SUBAPPLICATION logiBUS_AI_Calibrate_Remote_IDA_OPC (* 2-Punkt-Kalibrierung (AR_CALIBRATE_2P_REF, unabhaengig gespeicherte Rohwerte X_LOW/X_HIGH + Referenzwerte LOW_REF/HIGH_REF alle INI-persistiert) auf VT-Zahlenfelder (Rohwert + kalibrierter Wert, je eigene CNumberVariable) + Bargraph (kalibriert) + 2 VT-Tasten (CO/CS) + OPC-UA (Rohwert DWORD + kalibrierter Wert REAL, generisch, ein Kanal). Wie logiBUS_AI_Calibrate_IDA_OPC, aber der Rohwert kommt per Remote-Subscribe (AD_SUBSCRIBE_1) statt von einem lokalen logiBUS_AI_IDA - fuer Sensoren, deren physischer Analog-Eingang auf einer Station OHNE VT-Anschluss sitzt (z.B. Schnitthoehen-Winkelsensor B13 auf APIXON STG3, waehrend Kalibrierung+VT auf der Station mit VT-Anschluss laufen). Der Rohwert wird dort per logiBUS_AI_Raw_Publish_OPC publiziert. *)
  (* Standard: 61499-2; Description: Copyright (c) 2026 Meisterschulen am Ostbahnhof This program and the accompanying materials are made available under the terms of the Eclipse Public License 2.0 which is available at https://www.eclipse.org/legal/epl-2.0/ SPDX-License-Identifier: EPL-2.0 *)
  (* Version 1.0, 2026-09-12, Franz Höpfinger, Meisterschulen am Ostbahnhof, Remote-Rohwert-Variante von logiBUS_AI_Calibrate_IDA_OPC - logiBUS_AI_IDA+AD_SPLIT_2+AD_PUBLISH_RAW durch AD_SUBSCRIBE_1 ersetzt, Rest der Kalibrier-/VT-Kette unveraendert. Fuer Schnitthoehen-Winkelsensor B13 (STG3), Kalibrierung+VT auf STG1. *)
  (* Version 1.1, 2026-09-17, Franz Höpfinger, Meisterschulen am Ostbahnhof, AR_CALIBRATE_2P_REF.C_LOW/C_HIGH von AX-Sockets auf reine EventInputs umgestellt (Franz-Entscheidung, siehe logiBUS_AI_Calibrate_IDA_OPC v1.3) - AX_BOOL_TO_X_CO/_CS entfallen ersatzlos, E_MERGE_CO_B/E_MERGE_CS_B verbinden jetzt direkt per EventConnection mit CALIBRATE.C_LOW/C_HIGH. Dieser Typ ist ohnehin durch logiBUS_AI_Calibrated_Subscribe_VT_OPC (Analog-Lokal-Verarbeitung, Plan cuddly-bubbling-twilight) auf dem Weg zur Ablösung - Anpassung hier nur, damit die Datei weiterhin kompiliert. *)
  (* Version 1.2, 2026-09-18, Franz Höpfinger, Meisterschulen am Ostbahnhof, CO/CS-Merge-Ketten (2x E_MERGE_2 in Reihe) durch je einen einzelnen E_MERGE_3 ersetzt - OR-Merge ist assoziativ, funktional identisch. Siehe logiBUS_AI_Calibrate_IDA_OPC v1.4. *)
  (* Version 1.4, 2026-09-21, Franz Höpfinger, Meisterschulen am Ostbahnhof, Code-Review-Fund (PR #260): INI_X_HIGH.DEFAULT_VALUE stand auf REAL#1.0 statt 0.0 - AR_CALIBRATE_2P_REF's xHighCal-Kalibriert-Flag latchte dadurch bei JEDEM Boot sofort TRUE, obwohl HIGH nie kalibriert wurde. Default auf REAL#0.0 korrigiert. Betrifft Schnitthoehe/Oeltemperatur/Druck. *)
  (* Version 1.3, 2026-09-21, Franz Höpfinger, Meisterschulen am Ostbahnhof, AR_CALIBRATE_2P_REF hat jetzt ein INIT/QI/QO-Enable-Pattern (Bugfix Garbage-Interpolation bei nur einem kalibrierten Punkt + xClipping) - CALIBRATE bekommt Parameter QI=TRUE, sonst bleibt die FB im START-Zustand haengen und REQ laeuft nie. *)
  PACKAGE MyLib::sys;
  IMPORT isobus::UT::Q::const::IDs::ID_NULL;
  IMPORT logiBUS::utils::conversion::phys::NumericObjectPool_S;
  IMPORT isobus::UT::io::Button::ButtonActivationCode::BT_PRESSED_LATCHED;
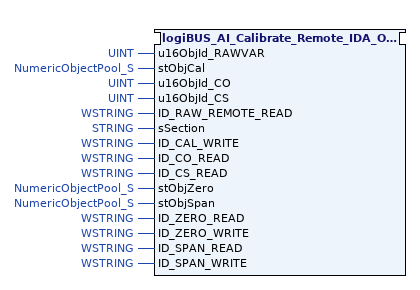
  VAR_INPUT
    u16ObjId_RAWVAR : UINT := ID_NULL; (* Object ID CNumberVariable (Rohwert 0-4095, unkalibriert, reine Diagnose-Anzeige) *)
    stObjCal : logiBUS::utils::conversion::phys::NumericObjectPool_S := (u16ObjId := ID_NULL, r32Scale := 1.0, i32Offset := 0, u8Decimals := 1); (* Object ID + Scale/Offset/Decimals CNumberVariable (kalibrierter Wert, eigene, unabhaengige CNumberVariable) *)
    u16ObjId_CO : UINT := ID_NULL; (* Object ID Taste 'CO' (Kalibrier-Nullpunkt: Referenz 1 anlegen, dann druecken) *)
    u16ObjId_CS : UINT := ID_NULL; (* Object ID Taste 'CS' (Kalibrier-Spanne: Referenz 2 anlegen, dann druecken - erst nach CO moeglich) *)
    ID_RAW_REMOTE_READ : WSTRING; (* Remote-Subscribe-Adresse des Rohwerts (DWORD 0-4095, ACTION=SUBSCRIBE) - Gegenstueck zu ID_RAW_WRITE auf der Sensor-Station (logiBUS_AI_Raw_Publish_OPC) *)
    sSection : STRING; (* INI-Sektionsname fuer X_LOW/X_HIGH/LOW_REF/HIGH_REF-Persistenz - pro Kanal eindeutig, sonst kollidieren die Kanaele in settings.ini *)
    ID_CAL_WRITE : WSTRING; (* Kalibrierter-Wert-Ruckmelde-Adresse (REAL, ACTION=PUBLISH) *)
    ID_CO_READ : WSTRING; (* Remote-CO-Adresse (BOOL, ACTION=SUBSCRIBE, togglet Kalibrier-Nullpunkt-Trigger wie ein Tastendruck - Web-Client schreibt bei jedem Klick den invertierten letzten Wert, jede Flanke (steigend ODER fallend) loest CO aus) *)
    ID_CS_READ : WSTRING; (* Remote-CS-Adresse (BOOL, ACTION=SUBSCRIBE, togglet Kalibrier-Spanne-Trigger wie ein Tastendruck - siehe ID_CO_READ) *)
    stObjZero : logiBUS::utils::conversion::phys::NumericObjectPool_S := (u16ObjId := ID_NULL, r32Scale := 1.0, i32Offset := 0, u8Decimals := 1); (* Object ID + Scale/Offset/Decimals CNumberVariable (ZERO-Referenzwert, VT-Eingabefeld + OPC-UA) *)
    stObjSpan : logiBUS::utils::conversion::phys::NumericObjectPool_S := (u16ObjId := ID_NULL, r32Scale := 1.0, i32Offset := 0, u8Decimals := 1); (* Object ID + Scale/Offset/Decimals CNumberVariable (SPAN-Referenzwert, VT-Eingabefeld + OPC-UA) *)
    ID_ZERO_READ : WSTRING; (* Remote-Subscribe-Adresse ZERO-Referenzwert (REAL, ACTION=SUBSCRIBE) *)
    ID_ZERO_WRITE : WSTRING; (* Remote-Echo-Adresse ZERO-Referenzwert (REAL, ACTION=PUBLISH) *)
    ID_SPAN_READ : WSTRING; (* Remote-Subscribe-Adresse SPAN-Referenzwert (REAL, ACTION=SUBSCRIBE) *)
    ID_SPAN_WRITE : WSTRING; (* Remote-Echo-Adresse SPAN-Referenzwert (REAL, ACTION=PUBLISH) *)
  END_VAR
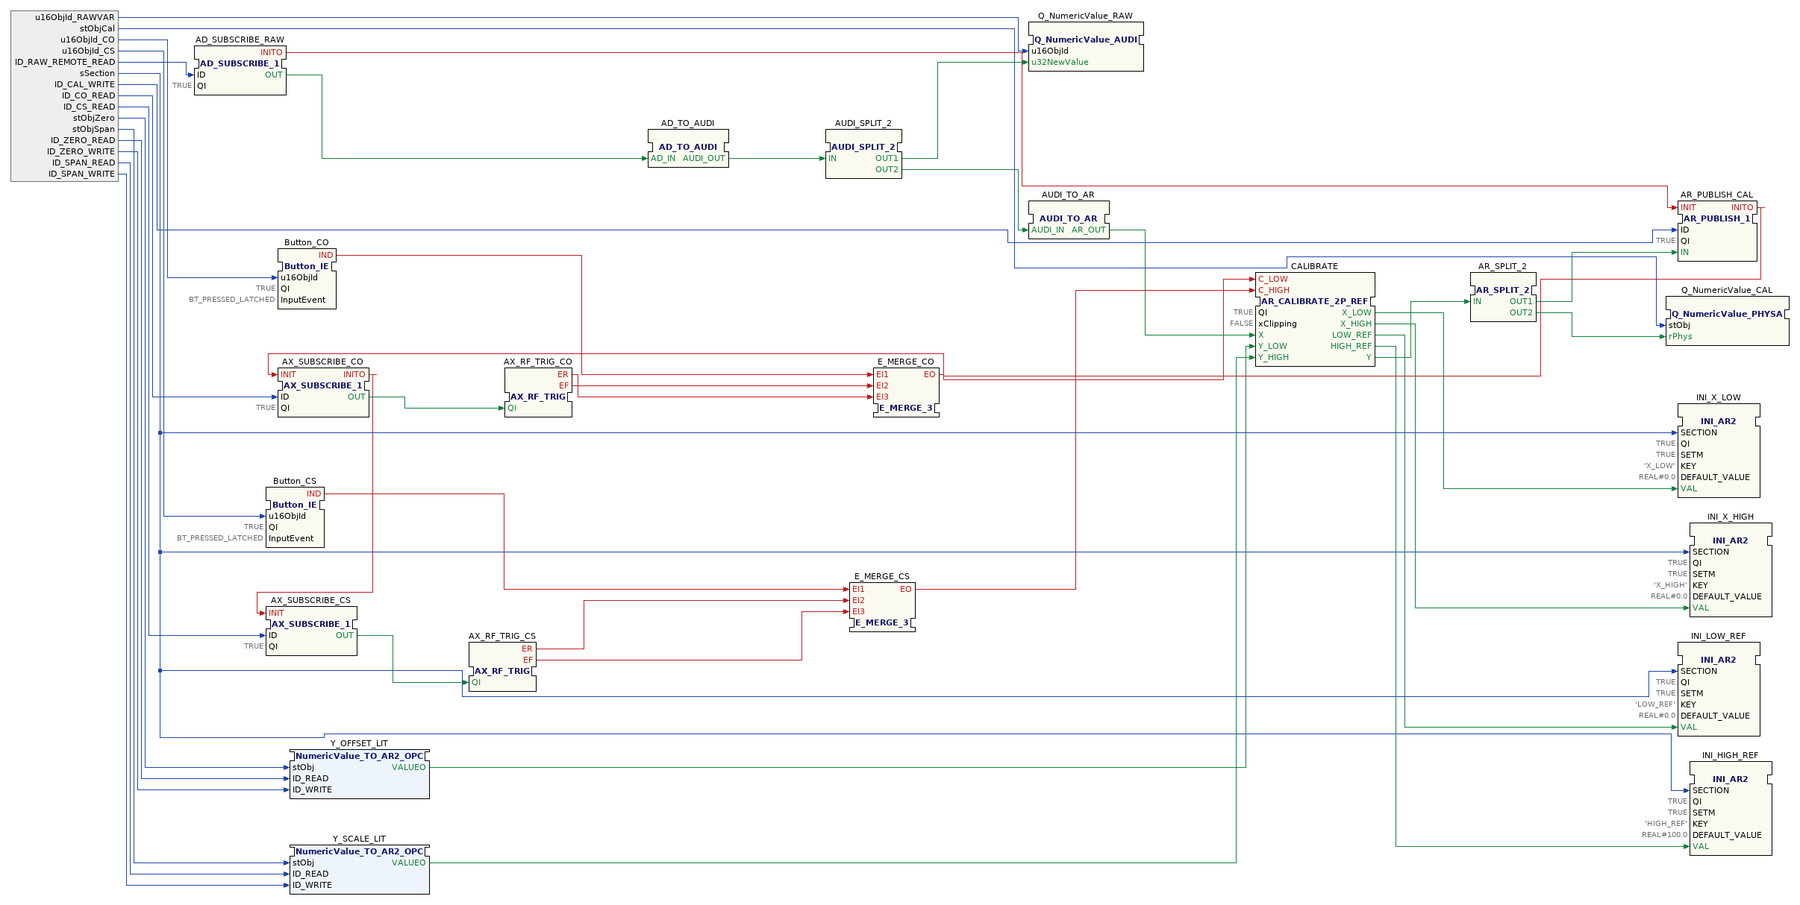
  FBS
    AD_SUBSCRIBE_RAW : adapter::net::AD_SUBSCRIBE_1(QI := TRUE);
    AD_TO_AUDI : adapter::conversion::unidirectional::AD_TO_AUDI;
    AUDI_SPLIT_2 : adapter::events::unidirectional::AUDI_SPLIT_2;
    Q_NumericValue_RAW : isobus::UT::Q::Q_NumericValue_AUDI;
    AUDI_TO_AR : adapter::conversion::unidirectional::AUDI_TO_AR;
    CALIBRATE : adapter::Engineering::measurements::AR_CALIBRATE_2P_REF(QI := TRUE, xClipping := FALSE);
    Button_CO : isobus::UT::io::Button::Button_IE(QI := TRUE, InputEvent := BT_PRESSED_LATCHED);
    Button_CS : isobus::UT::io::Button::Button_IE(QI := TRUE, InputEvent := BT_PRESSED_LATCHED);
    AX_SUBSCRIBE_CO : adapter::net::AX_SUBSCRIBE_1(QI := TRUE);
    AX_RF_TRIG_CO : adapter::events::unidirectional::AX_RF_TRIG;
    E_MERGE_CO : iec61499::events::E_MERGE_3;
    AX_SUBSCRIBE_CS : adapter::net::AX_SUBSCRIBE_1(QI := TRUE);
    AX_RF_TRIG_CS : adapter::events::unidirectional::AX_RF_TRIG;
    E_MERGE_CS : iec61499::events::E_MERGE_3;
    INI_X_LOW : eclipse4diac::storage::INI_AR2(QI := TRUE, SETM := TRUE, KEY := 'X_LOW', DEFAULT_VALUE := REAL#0.0);
    INI_X_HIGH : eclipse4diac::storage::INI_AR2(QI := TRUE, SETM := TRUE, KEY := 'X_HIGH', DEFAULT_VALUE := REAL#0.0);
    INI_LOW_REF : eclipse4diac::storage::INI_AR2(QI := TRUE, SETM := TRUE, KEY := 'LOW_REF', DEFAULT_VALUE := REAL#0.0);
    INI_HIGH_REF : eclipse4diac::storage::INI_AR2(QI := TRUE, SETM := TRUE, KEY := 'HIGH_REF', DEFAULT_VALUE := REAL#100.0);
    AR_SPLIT_2 : adapter::events::unidirectional::AR_SPLIT_2;
    AR_PUBLISH_CAL : adapter::net::AR_PUBLISH_1(QI := TRUE);
    Q_NumericValue_CAL : isobus::UT::Q::Q_NumericValue_PHYSA;
  END_FBS
  SUBAPPS
    Y_OFFSET_LIT : MyLib::sys::NumericValue_TO_AR2_OPC;
    Y_SCALE_LIT : MyLib::sys::NumericValue_TO_AR2_OPC;
  END_SUBAPPS
  EVENT_CONNECTIONS
    AD_SUBSCRIBE_RAW.INITO TO AR_PUBLISH_CAL.INIT;
    AR_PUBLISH_CAL.INITO TO AX_SUBSCRIBE_CO.INIT;
    AX_SUBSCRIBE_CO.INITO TO AX_SUBSCRIBE_CS.INIT;
    Button_CO.IND TO E_MERGE_CO.EI1;
    AX_RF_TRIG_CO.ER TO E_MERGE_CO.EI2;
    AX_RF_TRIG_CO.EF TO E_MERGE_CO.EI3;
    E_MERGE_CO.EO TO CALIBRATE.C_LOW;
    Button_CS.IND TO E_MERGE_CS.EI1;
    AX_RF_TRIG_CS.ER TO E_MERGE_CS.EI2;
    AX_RF_TRIG_CS.EF TO E_MERGE_CS.EI3;
    E_MERGE_CS.EO TO CALIBRATE.C_HIGH;
  END_CONNECTIONS
  DATA_CONNECTIONS
    u16ObjId_RAWVAR TO Q_NumericValue_RAW.u16ObjId;
    stObjCal TO Q_NumericValue_CAL.stObj;
    u16ObjId_CO TO Button_CO.u16ObjId;
    u16ObjId_CS TO Button_CS.u16ObjId;
    sSection TO INI_X_LOW.SECTION;
    sSection TO INI_X_HIGH.SECTION;
    sSection TO INI_LOW_REF.SECTION;
    sSection TO INI_HIGH_REF.SECTION;
    ID_RAW_REMOTE_READ TO AD_SUBSCRIBE_RAW.ID;
    ID_CAL_WRITE TO AR_PUBLISH_CAL.ID;
    ID_CO_READ TO AX_SUBSCRIBE_CO.ID;
    ID_CS_READ TO AX_SUBSCRIBE_CS.ID;
    stObjZero TO Y_OFFSET_LIT.stObj;
    ID_ZERO_READ TO Y_OFFSET_LIT.ID_READ;
    ID_ZERO_WRITE TO Y_OFFSET_LIT.ID_WRITE;
    stObjSpan TO Y_SCALE_LIT.stObj;
    ID_SPAN_READ TO Y_SCALE_LIT.ID_READ;
    ID_SPAN_WRITE TO Y_SCALE_LIT.ID_WRITE;
  END_CONNECTIONS
  ADAPTER_CONNECTIONS
    AD_SUBSCRIBE_RAW.OUT TO AD_TO_AUDI.AD_IN;
    AD_TO_AUDI.AUDI_OUT TO AUDI_SPLIT_2.IN;
    AUDI_SPLIT_2.OUT1 TO Q_NumericValue_RAW.u32NewValue;
    AUDI_SPLIT_2.OUT2 TO AUDI_TO_AR.AUDI_IN;
    AUDI_TO_AR.AR_OUT TO CALIBRATE.X;
    CALIBRATE.X_LOW TO INI_X_LOW.VAL;
    CALIBRATE.X_HIGH TO INI_X_HIGH.VAL;
    CALIBRATE.LOW_REF TO INI_LOW_REF.VAL;
    CALIBRATE.HIGH_REF TO INI_HIGH_REF.VAL;
    Y_OFFSET_LIT.VALUEO TO CALIBRATE.Y_LOW;
    Y_SCALE_LIT.VALUEO TO CALIBRATE.Y_HIGH;
    CALIBRATE.Y TO AR_SPLIT_2.IN;
    AR_SPLIT_2.OUT1 TO AR_PUBLISH_CAL.IN;
    AR_SPLIT_2.OUT2 TO Q_NumericValue_CAL.rPhys;
    AX_SUBSCRIBE_CO.OUT TO AX_RF_TRIG_CO.QI;
    AX_SUBSCRIBE_CS.OUT TO AX_RF_TRIG_CS.QI;
  END_CONNECTIONS
END_SUBAPPLICATION
